TYPE ST_Components_HMI_View :
STRUCT
END_STRUCT
END_TYPE

(* stored: Version 1.1.0.1
   DUT ST_Components_HMI_View: Id {b1dbc409-9cb2-0c37-3025-8079e0c639f8} *)
